// TIA Portal V20 export
DATA_BLOCK "Config"   // DB161
// stored: Access Published, MemoryReserve 100, Namespace Unit1.Em3
   VAR
      em : "LAF_typeEmConfiguration";   // Configuration of EM Parameters
      axis : Array[0.._.U1EM3_NO_OF_AXES] of DB_ANY;
      cmTopTapeJRDetect : "LBC_typeDigitalSignalConfiguration";
      cmTopTapeDiameter : "LBC_typeDigitalSignalConfiguration";
   END_VAR
   VAR RETAIN
      cmTopTapeAxisX : "LBC_typeAxis64PosConfiguration";
      cmTopTapeAxisY : "LBC_typeAxis64PosConfiguration";
   END_VAR
   VAR
      cmTopTapeLoadingBwdFwd : "LBC_typeTwoWayActuatorConfiguration";
      cmTopTapeLoadingClampOpenClose : "LBC_typeTwoWayActuatorConfiguration";
      cmTopTapeCutterUpDown : "LBC_typeTwoWayActuatorConfiguration";
      cmTopTapeCutterClampUpDown : "LBC_typeTwoWayActuatorConfiguration";
      cmTopTapeTensionBwdFwd : "LBC_typeTwoWayActuatorConfiguration";
      cmTopTapeAttachmentUpDown : "LBC_typeTwoWayActuatorConfiguration";
      cmTopTapeClampTopLeftUpDown : "LBC_typeTwoWayActuatorConfiguration";
      cmTopTapeClampTopCenterUpDown : "LBC_typeTwoWayActuatorConfiguration";
      cmTopTapeClampTopRightUpDown : "LBC_typeTwoWayActuatorConfiguration";
      cmTopTapeClampBtmDownUp : "LBC_typeTwoWayActuatorConfiguration";
      cmTopTapeClampAllOpenClose : "LBC_typeTwoWayActuatorConfiguration";
      cmTopTapeAttachmentVaccumOffOn : "LBC_typeTwoWayActuatorConfiguration";
      cmQrHandyReader : "LER_typeDM8700Configuration";
      softcam : Struct
         topTapeAxisX : "LER_typeSoftCamInterface";
         topTapeAxisY : "LER_typeSoftCamInterface";
      END_STRUCT;
   END_VAR
BEGIN
   em.referenceDesignator.parent := WSTRING#'U1';
   em.referenceDesignator.relative := WSTRING#'EM1';
   cmTopTapeAxisX.referenceDesignator := WSTRING#'TOP TAPING X-Axis';
   cmTopTapeAxisX.disableAlarms := FALSE;
   cmTopTapeAxisX.masterControlPopUp := TRUE;
   cmTopTapeAxisX.setPositions[0].position := 0.0;
   cmTopTapeAxisX.setPositions[1].position := 424.0;
   cmTopTapeAxisX.setPositions[3].position := 200.0;
   cmTopTapeAxisX.setPositions[0..1].velocity := 10.0;
   cmTopTapeAxisX.setPositions[3].velocity := 10.0;
   cmTopTapeAxisX.setPositions[0..1].acceleration := 100.0;
   cmTopTapeAxisX.setPositions[3].acceleration := 100.0;
   cmTopTapeAxisX.setPositions[0..1].deceleration := 100.0;
   cmTopTapeAxisX.setPositions[3].deceleration := 100.0;
   cmTopTapeAxisX.setPositions[0]."name" := 'Wait [Tape Get]';
   cmTopTapeAxisX.setPositions[1]."name" := 'Tape1 Put';
   cmTopTapeAxisX.setPositions[3]."name" := 'Remain Attachment';
   cmTopTapeAxisY.referenceDesignator := WSTRING#'TOP TAPING Y-Axis';
   cmTopTapeLoadingBwdFwd.referenceDesignator := WSTRING#'T.TAPE LOADING';
   cmTopTapeLoadingBwdFwd.monitoringDiscrepancy := T#5s;
   cmTopTapeLoadingClampOpenClose.referenceDesignator := WSTRING#'T.TAPE LOADING CLAMP';
   cmTopTapeLoadingClampOpenClose.monitoringDiscrepancy := T#5s;
   cmTopTapeCutterUpDown.referenceDesignator := WSTRING#'T.TAPE CUTTER';
   cmTopTapeCutterUpDown.monitoringDiscrepancy := T#5s;
   cmTopTapeCutterClampUpDown.referenceDesignator := WSTRING#'T.TAPE CUTTER CLAMP';
   cmTopTapeCutterClampUpDown.monitoringDiscrepancy := T#5s;
   cmTopTapeTensionBwdFwd.referenceDesignator := WSTRING#'T.TAPE TENSION';
   cmTopTapeTensionBwdFwd.monitoringDiscrepancy := T#5s;
   cmTopTapeAttachmentUpDown.referenceDesignator := WSTRING#'T.TAPE ATTACHMENT';
   cmTopTapeAttachmentUpDown.monitoringDiscrepancy := T#5s;
   cmTopTapeClampTopLeftUpDown.referenceDesignator := WSTRING#'T.TAPE CLAMP TOP LEFT';
   cmTopTapeClampTopLeftUpDown.monitoringDiscrepancy := T#5s;
   cmTopTapeClampTopCenterUpDown.referenceDesignator := WSTRING#'T.TAPE CLAMP TOP CENTER';
   cmTopTapeClampTopCenterUpDown.monitoringDiscrepancy := T#5s;
   cmTopTapeClampTopRightUpDown.referenceDesignator := WSTRING#'T.TAPE CLAMP TOP';
   cmTopTapeClampTopRightUpDown.monitoringDiscrepancy := T#5s;
   cmTopTapeClampBtmDownUp.referenceDesignator := WSTRING#'T.TAPE CLAMP BTM';
   cmTopTapeClampBtmDownUp.monitoringDiscrepancy := T#5s;
   cmTopTapeClampAllOpenClose.referenceDesignator := WSTRING#'TOP CLAMP ALL';
   cmTopTapeClampAllOpenClose.monitoringDiscrepancy := T#5s;
   cmTopTapeAttachmentVaccumOffOn.referenceDesignator := WSTRING#'ATTACHMENT VACUUM';
   cmTopTapeAttachmentVaccumOffOn.monitoringDiscrepancy := T#5s;
END_DATA_BLOCK
